Staubli VAL3: camera.pjx

Parameters version=s7.3.1 stackSize=5000 millimeterUnit=true
Program file=start.pgx
Program file=stop.pgx
Data file=camera.dtx
